FUNCTION_BLOCK SUBSCRIBE_1
  (* Description: Copyright (c) 2017 fortiss GmbH This program and the accompanying materials are made available under the terms of the Eclipse Public License 2.0 which is available at https://www.eclipse.org/legal/epl-2.0/ SPDX-License-Identifier: EPL-2.0 *)
  (* Version 1.0, 2017-10-25, Alois Zoitl, fortiss GmbH, initial API and implementation and/or initial documentation *)
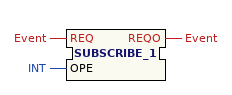
  EVENT_INPUT
    REQ;
  END_EVENT
  EVENT_OUTPUT
    REQO;
  END_EVENT
  VAR_INPUT
    OPE : INT;
  END_VAR
END_FUNCTION_BLOCK
